TYPE ST_CX_AdapterInfo :
STRUCT
	bDefault			: BOOL;
	strAdapterName		: STRING(75);
	bDHCPEnabled		: BOOL;
	strIPAddress		: T_IPv4Addr;
	strSubnetMask		: T_IPv4Addr;
	strDefaultGateway	: T_IPv4Addr;
END_STRUCT
END_TYPE

(* stored: Version 1.1.0.1
   DUT ST_CX_AdapterInfo: Id {80e66d5b-0390-4585-9d9b-cb3861cd82fc} *)
